{attribute 'qualified_only'}
{attribute 'strict'}
TYPE ENUM_EpicsMotorCmd :
	// Defines valid EPICS commands for nCommand
	// Copy from lcls-twincat-motion PR#31
(
	JOG := 0,
	MOVE_VELOCITY := 1,
	MOVE_RELATIVE := 2,
	MOVE_ABSOLUTE := 3,
	MOVE_MODULO := 4,
	HOME := 10,
	GEAR := 30
);
END_TYPE

(* stored: Version 1.1.0.1, ProductVersion 3.1.4022.18
   DUT ENUM_EpicsMotorCmd: Id {6aeca57a-6008-439f-9ea1-66c05e3b253c} *)
